FUNCTION_BLOCK DelayedAddCommand EXTENDS AddCommand
VAR
	fbTonDelay		: TON;
END_VAR

// OO-Class 
SUPER^();

METHOD PROTECTED CalculateProgress
IF stHandshake.nResultCode = 99 OR stHandshake.nResultCode = E_CommandResultCode.Done THEN
	stHandshake.nProgress := 100;
ELSE
	stHandshake.nProgress := REAL_TO_BYTE(100.0 / TIME_TO_REAL(fbTonDelay.PT) * TIME_TO_REAL(fbTonDelay.ET));
END_IF
END_METHOD

METHOD Protected Cancelled
SUPER^.Cancelled();

// Reset Input for next start
fbTonDelay(IN:=stHandshake.bBusy);

// Set result to invalid value
Result := -1;
END_METHOD

METHOD PROTECTED Done
SUPER^.Done();

// Reset Input for next start
fbTonDelay(IN:=stHandshake.bBusy);
END_METHOD

METHOD FB_init : BOOL
VAR_INPUT
	bInitRetains 		: BOOL; 		// if TRUE, the retain variables are initialized (warm start / cold start)
	bInCopyCode 		: BOOL;  		// if TRUE, the instance afterwards gets moved into the copy code (online change)
	tDelayTime 			: TIME;			// Time to deleay the Running state
END_VAR
fbTonDelay.PT := tDelayTime;
END_METHOD

METHOD PROTECTED Task : BOOL
fbTonDelay(IN:=stHandshake.bBusy);

IF fbTonDelay.Q THEN
	// Execute base Task in AddCommand for Addition
	SUPER^.Task();
	
	// Exection is finished, set nResultCode = 99
	
	Finish(E_CommandResultCode.Done);
END_IF
END_METHOD

END_FUNCTION_BLOCK

(* stored: Version 1.1.0.1, ProductVersion 3.1.4022.10
   POU DelayedAddCommand: Id {65b2ca40-9e7e-4cdc-82b9-f7b2c503faa2}, SpecialFunc None
   Method CalculateProgress: Id {5cea9727-992d-40c4-9429-66e19c9b7a56}
   Method Cancelled: Id {5607005d-a3e2-4a0d-8acf-89dd886f9689}
   Method Done: Id {d3f67563-493c-480a-88ee-d8edb11f7e53}
   Method FB_init: Id {36cce40c-7f51-0818-1bf9-386ad9ff80ee}
   Method Task: Id {7c566ce4-fa9b-444f-bb18-8e5071761b78} *)
